// Mitsubishi GX Works2 project: 250916_A+A-B+B-C+C- 반복 - 복사본   PLC: Q02U

PROGRAM MAIN
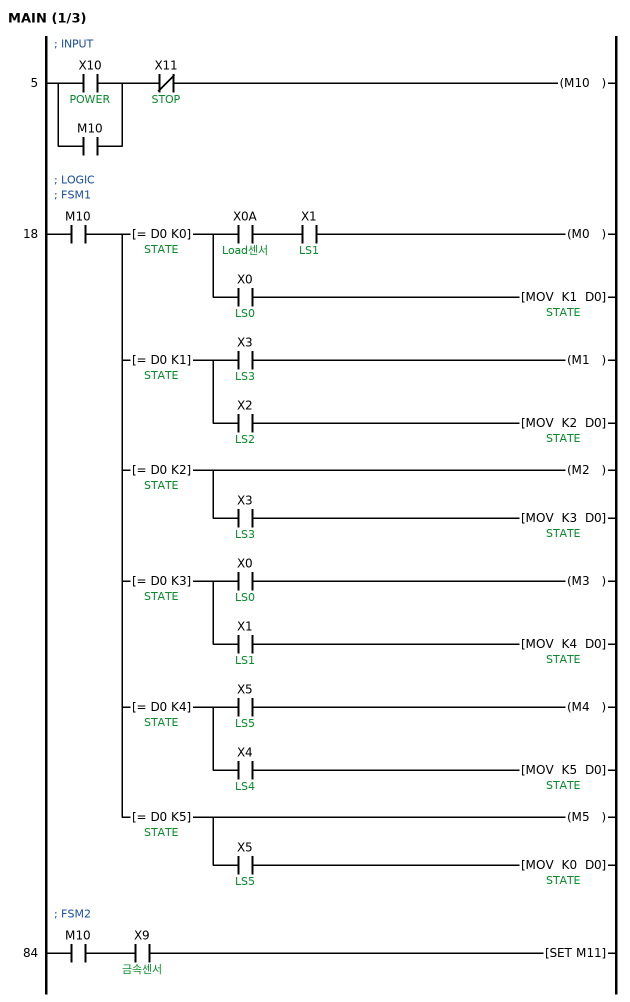
; INPUT
5     LD      X10  ; POWER
      OR      M10
      ANI     X11  ; STOP
      OUT     M10
; LOGIC
; FSM1
18    LD      M10
      MPS
      AND=    D0 K0  ; STATE
      MPS
      AND     X0A  ; Load센서
      AND     X1  ; LS1
      OUT     M0
      MPP
      AND     X0  ; LS0
      MOV     K1 D0
      MRD
      AND=    D0 K1  ; STATE
      MPS
      AND     X3  ; LS3
      OUT     M1
      MPP
      AND     X2  ; LS2
      MOV     K2 D0
      MRD
      AND=    D0 K2  ; STATE
      OUT     M2
      AND     X3  ; LS3
      MOV     K3 D0
      MRD
      AND=    D0 K3  ; STATE
      MPS
      AND     X0  ; LS0
      OUT     M3
      MPP
      AND     X1  ; LS1
      MOV     K4 D0
      MRD
      AND=    D0 K4  ; STATE
      MPS
      AND     X5  ; LS5
      OUT     M4
      MPP
      AND     X4  ; LS4
      MOV     K5 D0
      MPP
      AND=    D0 K5  ; STATE
      OUT     M5
      AND     X5  ; LS5
      MOV     K0 D0
; FSM2
84    LD      M10
      AND     X9  ; 금속센서
      SET     M11
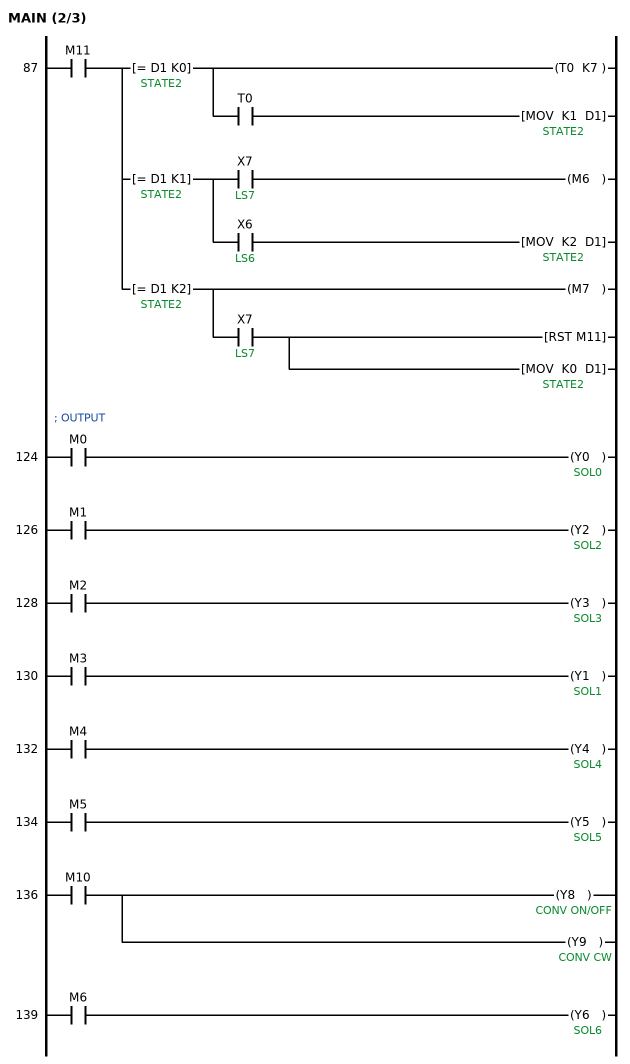
87    LD      M11
      MPS
      AND=    D1 K0  ; STATE2
      OUT     T0 K7
      AND     T0
      MOV     K1 D1
      MRD
      AND=    D1 K1  ; STATE2
      MPS
      AND     X7  ; LS7
      OUT     M6
      MPP
      AND     X6  ; LS6
      MOV     K2 D1
      MPP
      AND=    D1 K2  ; STATE2
      OUT     M7
      AND     X7  ; LS7
      RST     M11
      MOV     K0 D1
; OUTPUT
124   LD      M0
      OUT     Y0  ; SOL0
126   LD      M1
      OUT     Y2  ; SOL2
128   LD      M2
      OUT     Y3  ; SOL3
130   LD      M3
      OUT     Y1  ; SOL1
132   LD      M4
      OUT     Y4  ; SOL4
134   LD      M5
      OUT     Y5  ; SOL5
136   LD      M10
      OUT     Y8  ; CONV ON/OFF
      OUT     Y9  ; CONV CW
139   LD      M6
      OUT     Y6  ; SOL6
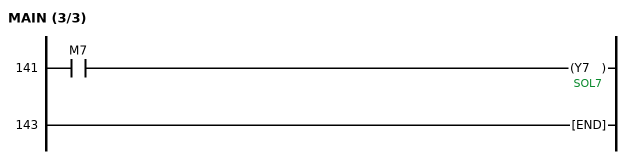
141   LD      M7
      OUT     Y7  ; SOL7
143   END
END_PROGRAM

// device comments not shown above
X8  ; 근접센서
Y0A  ; CONV CCW
Y0B  ; RED LAMP
Y0C  ; YELLOW LAMP
Y0D  ; GREEN LAMP
